FUNCTION_BLOCK ABSTRACT Timer_Abstract IMPLEMENTS I_Timer
VAR_INPUT
END_VAR
VAR_OUTPUT
END_VAR
VAR
	_Setting 	: ST_Setting;
	_Input 		: ST_Input;
	_Output     : ST_Output;
END_VAR


PROPERTY Input : REFERENCE TO ST_Input
SET
THIS^._Input := Input;
END_SET
END_PROPERTY


PROPERTY Output : REFERENCE TO ST_Output
GET
Output REF= THIS^._Output;
END_GET
END_PROPERTY


METHOD ABSTRACT Run
END_METHOD


PROPERTY Setting : REFERENCE TO ST_Setting
SET
THIS^._Setting := Setting;
END_SET
END_PROPERTY

END_FUNCTION_BLOCK

(* stored: Version 1.1.0.1, ProductVersion 3.1.4024.12
   POU Timer_Abstract: Id {16764f21-872a-4462-b20e-5c4063cdd38a}, SpecialFunc None
   Property Input: Id {ea075b2c-1a90-470d-a0b7-01d39144eb2a}
   Set Set: Id {323678a0-addf-419c-935f-8a249a8b1fb3}
   Property Output: Id {934d7402-5635-41b7-a552-e617723f545b}
   Get Get: Id {0e6781db-9c98-4dbe-b9d7-f89b709ece3e}
   Method Run: Id {10b4d269-36ed-46c3-8ffe-df48d8149806}
   Property Setting: Id {b6984b6d-bfcd-4204-98b3-9eb2fc47202f}
   Set Set: Id {f3c93a8a-e125-444e-8bba-600f5e90645f} *)
